{attribute 'qualified_only'}
//{attribute 'strict'}
{attribute 'to_string'}
TYPE E_INSTANCE_STATE :
(
  NULL,
	INVALID,
  INIT,
  DISABLED,
  DETECTION,
  ENABLED,
  WORKING,
  PROCEEDING,
  FINISH,
  CLEARED
)UINT;
END_TYPE

(* stored: Version 1.1.0.1
   DUT E_INSTANCE_STATE: Id {33f09526-67e0-4b76-b2c8-159a1d81e8b2} *)
